Fanuc KAREL source: ks00006.KL

PROGRAM KS00006
%STACKSIZE=65535
%PRIORITY=65535
%NOLOCKGROUP
TYPE
REC_T=STRUCTURE
VALUE : INTEGER
FLAG : BOOLEAN
ENDSTRUCTURE
VAR
A : REC_T
B : REC_T
FLAG : BOOLEAN
N : INTEGER
STATUS : INTEGER
PN : STRING[80]
VN : STRING[80]
BEGIN
PN=''
VN='A'
-- UNRESOLVED_PC line 19 opcodes [27 22 22 2A 22 2A 22 22 AF] marker_code=27
END KS00006
